PROGRAM F_FactoryIO_Read_Inputs
VAR;
	LFB_MBReadInputs 	: FB_MBReadInputs;
END_VAR

LFB_MBReadInputs(
	sIPAddr := '127.0.0.1',
	nTCPPort := 505,
	nUnitID := 255,
	nQuantity := 16,
	nMBAddr := 0,
	cbLength := SIZEOF(GAB_FactoryIO_Inputs),
	pDestAddr := ADR(GAB_FactoryIO_Inputs),
	bExecute := TRUE,
	tTimeout := T#1S,
	bBusy => ,
	bError => ,
	nErrId => ,
	cbRead => ,
 );
LFB_MBReadInputs(bExecute := FALSE);

END_PROGRAM

(* stored: Version 1.1.0.1, ProductVersion 3.1.4024.4
   POU F_FactoryIO_Read_Inputs: Id {af80393c-eb61-4b06-bd54-a00a692f53f7}, SpecialFunc None *)
